FUNCTION_BLOCK Overcurrent_Protector (* Extracted Composite Function Block Type *)
  (* Standard: 61499-2 *)
  (* Version 1/31/2024, Maxth *)
  PACKAGE Main;
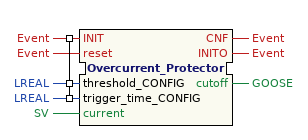
  EVENT_INPUT
    INIT WITH threshold_CONFIG, trigger_time_CONFIG;
    reset;
  END_EVENT
  EVENT_OUTPUT
    CNF;
    INITO;
  END_EVENT
  VAR_INPUT
    threshold_CONFIG : LREAL;
    trigger_time_CONFIG : LREAL;
  END_VAR
  SOCKETS
    current : SV;
  END_SOCKETS
  PLUGS
    cutoff : GOOSE;
  END_PLUGS
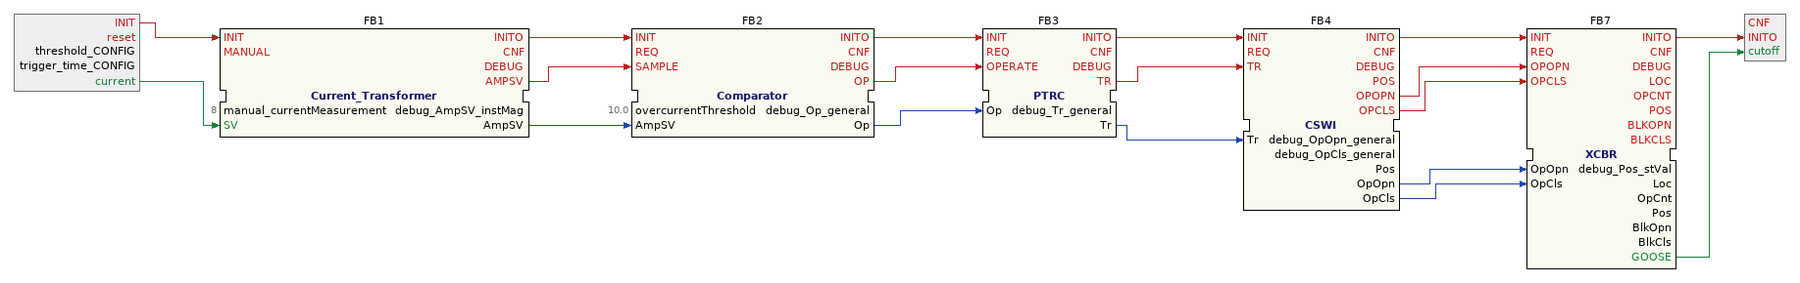
  FBS
    FB1 : Current_Transformer(manual_currentMeasurement := 8);
    FB2 : Comparator(overcurrentThreshold := 10.0);
    FB3 : PTRC;
    FB4 : CSWI;
    FB7 : XCBR;
  END_FBS
  EVENT_CONNECTIONS
    FB1.INITO TO FB2.INIT;
    FB1.AMPSV TO FB2.SAMPLE;
    FB2.INITO TO FB3.INIT;
    FB2.OP TO FB3.OPERATE;
    FB3.INITO TO FB4.INIT;
    FB3.TR TO FB4.TR;
    FB4.INITO TO FB7.INIT;
    FB4.OPOPN TO FB7.OPOPN;
    FB4.OPCLS TO FB7.OPCLS;
    INIT TO FB1.INIT;
    FB7.INITO TO INITO;
  END_CONNECTIONS
  DATA_CONNECTIONS
    FB1.AmpSV TO FB2.AmpSV;
    FB2.Op TO FB3.Op;
    FB3.Tr TO FB4.Tr;
    FB4.OpOpn TO FB7.OpOpn;
    FB4.OpCls TO FB7.OpCls;
  END_CONNECTIONS
  ADAPTER_CONNECTIONS
    current TO FB1.SV;
    FB7.GOOSE TO cutoff;
  END_CONNECTIONS
END_FUNCTION_BLOCK
